FUNCTION_BLOCK SHL_BYTE (* See SHIFT_ANY *)
  (* Standard: 61131-3 *)
  (* Version 0.1, 2006-09-09, JHC, Holobloc Inc, Converted to Template. *)
  (* Version 0.0, 2004-12-15, JHC, Rockwell Automation, Converted from SRC format. *)
  (* Compiler header: package fb.rt.plc.bits; *)
  (* Compiler classdef: (IN << N) *)
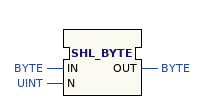
  VAR_INPUT
    IN : BYTE;
    N : UINT;
  END_VAR
  VAR_OUTPUT
    OUT : BYTE;
  END_VAR
END_FUNCTION_BLOCK
